(* Base of Module Sequences. Inheriting FBs must provide the main implementation. *)
FUNCTION_BLOCK ABSTRACT ModuleSequenceBase EXTENDS BehaviorBase
VAR
	m_ptrProcessManager: POINTER TO ProcessManager;
	m_ptrStateTracker: POINTER TO StateTracker;
END_VAR

METHOD ProvideServices : BOOL
VAR_INPUT
	i_ptrProcessManager: POINTER TO ProcessManager;
	i_ptrStateTracker: POINTER TO StateTracker;
END_VAR
THIS^.m_ptrProcessManager := i_ptrProcessManager;
THIS^.m_ptrStateTracker := i_ptrStateTracker;
END_METHOD

METHOD RequestRecovery : BOOL
VAR_INPUT
END_VAR
THIS^.m_ptrProcessManager^.RequestRecovery(THIS^.Postcondition, TO_STRING(m_id));
END_METHOD

END_FUNCTION_BLOCK

(* stored: Version 1.1.0.1
   POU ModuleSequenceBase: Id {d9e2fd9d-c089-4bdc-9e23-2df4eba13108}, SpecialFunc None
   Method ProvideServices: Id {c6a37104-0206-492a-8d30-fb08e3ab0d97}
   Method RequestRecovery: Id {a831c301-ba78-45b4-b05a-093ad147011c} *)
